TYPE "udtRoomAI"
VERSION : 0.1
   STRUCT
      IW_RoomTemperature_1 { ExternalAccessible := 'False'; ExternalVisible := 'False'; ExternalWritable := 'False'} : Int;
      IW_RoomHumidity_1 { ExternalAccessible := 'False'; ExternalVisible := 'False'; ExternalWritable := 'False'} : Int;
   END_STRUCT;

END_TYPE

